(* CODESYS project CtaSysInfluxLog_2.0.0.1.library
   Description: Trendlog Library der CTA
   Version: 2.0.0.1
   Title: CtaSysInfluxLog
   Author: SIS
   DocFormat: reStructuredText
   LanguageModelAttribute: qualified-access-only
   Placeholder: CtaSysInfluxLog
   CompiledLibraryCompatibilityVersion: CODESYS V3.5 SP16 Patch 3
   Company: CTA
   DefaultNamespace: CtaSysInfluxLog

Project tree, tasks and I/O mapping:
  libraries: Standard, 3.5.18.0 (System); VisuSymbols, 4.5.0.0 (System); CtaSysConfig, 2.0.0.0 (CTA); SysFile, 3.5.17.0 (System); SysProcess, 3.5.17.0 (System); StringUtils, 3.5.20.0 (System); CtaVisSymbols, 2.0.0.0 (CTA); CmpIecTask, 3.5.20.50 (System); Common Behaviour Model, 4.0.0.0 (CODESYS); Util, 3.5.19.0 (System); CmpErrors2 Interfaces, * (System); CmpEventMgr, 3.5.17.0 (System); CmpApp, 3.5.17.0 (System); SysDir, 3.5.17.0 (System); SysTypes Interfaces, * (System); CtaAppTime, 1.0.0.1 (CTA)
  40 Visualizations/
    visualisation visInfluxDb
    visualisation visInfluxDbTemp
    visualisation VIS_POPUP_INFLUXDB
  30 Program Organization Units/
    function block FB_INFLUX_LOG [ST]: SendData, FileClose, FileOpen, FileWrite, CreateDataBase, FileDelete, ADD_LOG_NODE, REM_LOG_NODE, DataBuffer, Config, CheckToBigFile, FB_INIT
    NODE/
      BASE/
        function block FB_LOG_NODE [ST]: KEY, VALUE, BIG_SYBIL, ENABLE, SELF, LOW_SYBIL, REGISTER, FB_EXIT, UNREGISTER, LOGTYPE, DESTROY, DESTROYAFTERLOG, UNIXTIME
      STRING/
        function block FB_LOG_NODE_STRING [ST]: SET_VALUE, VALUE, LOGTYPE
      BOOL/
        function block FB_LOG_NODE_BOOL [ST]: VALUE, SET_VALUE, LOGTYPE
      INT/
        function block FB_LOG_NODE_INT [ST]: VALUE, SET_VALUE, LOGTYPE
      REAL/
        function block FB_LOG_NODE_REAL [ST]: VALUE, SET_VALUE, LOGTYPE
    SPACE CATCH/
      function fcSpaceCatch [ST]
    ASYNC SEND/
      function block FB_SEND_ASYNC [ST]: StartAction, SendAction, ResetAction, FB_INIT, DropAction
    FACTORY/
      function block FB_NODE_FACTORY [ST]: GET_BOOL_LOG_NODE, GET_INT_LOG_NODE, GET_REAL_LOG_NODE, GET_STRING_LOG_NODE, READY
    TREND TASK/
      function block FB_TREND_TASK_PROVIDER [ST]: FB_INIT, FB_EXIT, EventCallback
    TASK_SCHEDULER/
      function CYCLIC_TRENDLOG_BACKGROUND_CTA [ST]
      function CYCLIC_TRENDLOG_CTA [ST]
    function GetWorkingDirectory [ST]
  00000000-0000-0000-0000-000000000000|D:\CoDeSys\LibrariesV3\trunk\Intern\CAA\CAA Template\3.4.0.0 draft\Placeholder.xml
  00000000-0000-0000-0000-000000000000|D:\CoDeSys\LibrariesV3\trunk\Intern\CAA\CAA Template\3.2.0.3 draft\Prefix.pdf
  00000000-0000-0000-0000-000000000000|D:\CoDeSys\LibrariesV3\trunk\Intern\CAA\CAA Template\3.5.2.0 draft\Placeholder.xml
  20 Structs/
    data type scParameter
  50 Images/
  10 Documenation/
    global variables VersionHistory
    global variables readMe
  21 Interface/
    interface ITF_LOG_NODE: BIG_SYBIL, KEY, VALUE, ENABLE, SELF, LOGTYPE, LOW_SYBIL, DESTROYAFTERLOG, DESTROY, UNIXTIME
    interface ITF_LOG_NODE_BOOL: SET_VALUE
    interface ITF_LOG_NODE_INT: SET_VALUE
    interface ITF_LOG_NODE_REAL: SET_VALUE
    interface ITF_LOG_NODE_STRING: SET_VALUE
  11 Library Parameter/
  12 Konstanten/
  60 Textlisten/
    text list InfluxStartup
    text list LogState
  13 Globale Variablen/
    global variables GVL_TREND
    global variables GVL_TREND_TASK_PROVIDER
  text list GlobalTextList
  22 Enumeration/
    data type enInfluxDataType
  70 PRG/
*)

// 20 Structs/scParameter
TYPE scParameter :
    STRUCT
       fbServerIp		:	CtaSysConfig.fbSTRING40;
		fbDataBase		:	CtaSysConfig.fbSTRING40;
		fbtLogIntervall	:	CtaSysConfig.fbTIME;
		fbxEnable		:	CtaSysConfig.fbBOOL;
		fbuiPort		:	CtaSysConfig.fbUINT;
    END_STRUCT
END_TYPE

// 22 Enumeration/enInfluxDataType
{attribute 'qualified_only'}
TYPE enInfluxDataType :
(
	TYPE_BOOL 	:= 0,
	TYPE_INT	:= 1,
	TYPE_REAL 	:= 2,
	TYPE_STRING	:= 3	
);
END_TYPE

// 10 Documenation/VersionHistory
(* 

.. image:: ../../Images/CTA_Logo.jpg
   :align: right
   :width: 15% 

**Vorlage**   


============ =========== =========== ============================================
**Date**     **Version** **Author**  **Change**
------------ ----------- ----------- --------------------------------------------
04.03.2021   0.0.0.0     SIS         Vorlage erstellt

============ =========== =========== ============================================


*)
VAR_GLOBAL
    stInfo : STRING:= '0.0.0.0, Vorlage, CTA';
END_VAR

// 10 Documenation/readMe
(*

**ReadMe**

|	**Empfehlung**
|
|	Für das Trendloggen in die InfluxDb wird nachfolgender Code benötigt.                           
|	Zusätzlich muss im PLC_PRG der Fb fbLibAp94_1InfluxDb als Funktionsbaustein Instanziert werden.
|  
|
| *Beispiel* 

 ============= ================================================================================================================================
 Beschreibung  Code                                                                                                
 ============= ================================================================================================================================                   
 Pou oder SmFb .. code-block:: codesys
 
                    // Deklaration der Struktur Variable scInfluxData
                    VAR
                        scInfluxData                    :   WagoAppInfluxDB.typInfluxField;
                    END_VAR     

                    (* Code als actInfluxDb *)
                    // Clear Data
                        scInfluxData.sKey   := '';
                        scInfluxData.sValue := '';
                    // Write Data
                        scInfluxData.sKey   := CONCAT(STR1 := stObjID, STR2 := '_xOn');
                        scInfluxData.sValue := TO_STRING(xOn); 
                        scInfluxData.eType  := WagoAppInfluxDB.eFieldValueType.eFVT_BOOL;
                        LibAp94InfluxDb.gvlLibAp94_1InfluxDb.fbLibAp94_2DataCollecter.proInfluxDbData := scInfluxData;
                    // Clear Data
                        scInfluxData.sKey   := '';
                        scInfluxData.sValue := '';
                    // Write Data
                        scInfluxData.sKey   := CONCAT(STR1 := stObjID, STR2 := '_rOnY');
                        scInfluxData.sValue := TO_STRING(rOnY); 
                        scInfluxData.eType  := WagoAppInfluxDB.eFieldValueType.eFVT_FLOAT;
                        LibAp94InfluxDb.gvlLibAp94_1InfluxDb.fbLibAp94_2DataCollecter.proInfluxDbData := scInfluxData;    
                    // Clear Data
                        scInfluxData.sKey   := '';
                        scInfluxData.sValue := '';
                    // Write Data
                        scInfluxData.sKey   := CONCAT(STR1 := stObjID, STR2 := '_xError');
                        scInfluxData.sValue := TO_STRING(proLockDown); 
                        scInfluxData.eType  := WagoAppInfluxDB.eFieldValueType.eFVT_BOOL;
                        LibAp94InfluxDb.gvlLibAp94_1InfluxDb.fbLibAp94_2DataCollecter.proInfluxDbData := scInfluxData;           
                                                                                                                                                                 
 ============= ================================================================================================================================ 
*)
VAR_GLOBAL
    xReadMeDone              :   BOOL;
END_VAR

// 13 Globale Variablen/GVL_TREND
{attribute 'qualified_only'}
{attribute 'linkalways'}
{attribute 'global_init_slot' := '1000'}
VAR_GLOBAL
	(* ASYNC SEND *)
	ASYNC_SEND				:	FB_SEND_ASYNC;	
	FB_INFLUX_LOG_OBJ		:	FB_INFLUX_LOG;
	FB_INFLUX_NODE_FACTORY	:	FB_NODE_FACTORY;
END_VAR

// 13 Globale Variablen/GVL_TREND_TASK_PROVIDER
{attribute 'qualified_only'}
{attribute 'linkalways'}
{attribute 'global_init_slot' := '1001'}
VAR_GLOBAL
	FB_TREND_TASK_PROVIDER_GLOBAL : FB_TREND_TASK_PROVIDER;	
	dwSEMA_CYCLIC	:	DWORD;				// CYCLIC TASK Semaphore
	dwSEMA_BACK		:	DWORD;				// BACKGRROUND TASK Semaphore
END_VAR

// 21 Interface/ITF_LOG_NODE
INTERFACE ITF_LOG_NODE EXTENDS __SYSTEM.IQueryinterface

PROPERTY BIG_SYBIL : ITF_LOG_NODE
GET
END_GET
SET
END_SET
END_PROPERTY

PROPERTY KEY : STRING(255)
GET
END_GET
SET
END_SET
END_PROPERTY

PROPERTY VALUE : STRING(255)
GET
END_GET
END_PROPERTY

PROPERTY ENABLE : BOOL
SET
END_SET
GET
END_GET
END_PROPERTY

PROPERTY SELF : ITF_LOG_NODE
GET
END_GET
END_PROPERTY

PROPERTY LOGTYPE : enInfluxDataType
GET
END_GET
END_PROPERTY

PROPERTY LOW_SYBIL : ITF_LOG_NODE
GET
END_GET
SET
END_SET
END_PROPERTY

PROPERTY DESTROYAFTERLOG : BOOL
SET
END_SET
GET
END_GET
END_PROPERTY

METHOD INTERNAL DESTROY
VAR_INPUT
END_VAR
END_METHOD

PROPERTY UNIXTIME : ULINT
GET
END_GET
END_PROPERTY

END_INTERFACE

// 30 Program Organization Units/FB_INFLUX_LOG
FUNCTION_BLOCK FB_INFLUX_LOG
VAR
	(* Server Info *)
	UNIXTIME		:	STRING(20);
	(* Log Nodes *)
	_BASE_LOG_NODE	:	ITF_LOG_NODE;
	_TEMP_REG_NODE	:	ITF_LOG_NODE;
	_TEMP_LOG_NODE	:	ITF_LOG_NODE;	
	_TEMP_DES_NODE	:	ITF_LOG_NODE;
	_COUNT			:	UINT;
	(* Case *)
	usiStartUpCase	:	USINT;
	usiLogCase		:	USINT;
	xAbort			:	BOOL;
	(* Buffer *)
	BUFFER			:	STRING(912);
	(* Timers *)
	DELAY			:	Standard.TON	:= (PT := T#20S);
	PULSE			:	Standard.TON	:= (PT := T#1S);
	Fb_TIME			:	CtaAppTime.fbTimeMeasurement;
	ltOut			:	LTIME;
	Fb_TIME_TO_BIG	:	CtaAppTime.fbTimeMeasurement;
	ltOutToBig		:	LTIME;
	xFirstToBig		:	BOOL;
	tCycle			:	TIME;
	taskHandle		:	SysTypes.RTS_IEC_HANDLE;
	pInfo 			: 	POINTER TO CmpIecTask.Task_Info2;	
	(* File Handling *)
	FILE_HANDLE		:	SysFile.RTS_IEC_HANDLE;
	RESULT			:	SysFile.RTS_IEC_RESULT;
	LASTBIGFILESIZE	:	__XWORD;
	FILE_PATH		:	STRING(255);
	(* Config *)
	fbConfigFile	:	CtaSysConfig.fbConfigFile;
	(* Parameter *)
	scParameter		:	scParameter;	
END_VAR
VAR CONSTANT
	COMMA		:	STRING[1] := ',';
	EQUAL		:	STRING[1] := '=';
	SPACE		:	STRING[1] := ' ';
	LINE		:	STRING[1] := '$N';
END_VAR

(* Config *)
Config();
(* Start Up Case *)
CASE usiStartUpCase OF
	0:	(* Delay *)
		DELAY(IN	:= fbConfigFile.proInitDone AND NOT DELAY.Q ,
			  PT	:= T#10S);
		(* Wait *)
		IF DELAY.Q AND scParameter.fbxEnable.proValue THEN
			(*  Get Cycle Time *)
			taskHandle :=  CmpIecTask.IecTaskGetCurrent(ADR(RESULT));
			IF taskHandle <> 0 THEN
				pInfo := CmpIecTask.IecTaskGetInfo3(taskHandle,ADR(RESULT));
				IF pInfo <> 0 THEN
					tCycle := TO_TIME(pInfo^.dwInterval/1000);
				END_IF;		
			END_IF;
			(* SERVER & DATABASE INFO *)
			GVL_TREND.ASYNC_SEND.SERVER 	:= scparameter.fbServerIp.proValue;
			GVL_TREND.ASYNC_SEND.DATABASE 	:= scparameter.fbDataBase.proValue;
			GVL_TREND.ASYNC_SEND.PORT		:= scparameter.fbuiPort.proValue;
			(* Next Case *)
			usiStartUpCase := usiStartUpCase + 1;	
		END_IF;
	1:	(* Create Database *)
		IF CreateDataBase() THEN
			usiStartUpCase := usiStartUpCase + 1;
			usiLogCase   := 1;
		ELSE
			usiStartUpCase := 0;	// Retray with case 0
		END_IF;
	2:	(* Log *)
		CASE usiLogCase OF
			0:
				(* Wait for Database*)
				usiLogCase := usiLogCase + 1;	
				(* ASYNC SEND RESET*)
				GVL_TREND.ASYNC_SEND.Execute := FALSE;		
			1:	
				(* Open File to Save Log *)
				FileOpen();
				usiLogCase := usiLogCase + 1;
			2:	
				(* Log Intervall *)
				PULSE(	IN	:= NOT PULSE.Q,	
						PT	:= LIMIT(T#0MS,scparameter.fbtLogIntervall.proValue - MIN(scparameter.fbtLogIntervall.proValue,(TO_TIME(ltOut)+(tCycle*4)+ T#500MS)),T#10M));

				(* Start Log *)
				IF PULSE.Q OR PULSE.PT = T#0MS THEN
					Fb_TIME.Start();
					UNIXTIME := CONCAT(TO_STRING(Util.GetLocalDateTime(Util.TSW.gc_tzTimeZoneUTC)),'000000');
					(* Get Active Log Data *)
					_COUNT := 0;
					IF __QUERYINTERFACE(_BASE_LOG_NODE,_TEMP_LOG_NODE) THEN
						REPEAT
							(* Check if Valid Log Node *)
							IF __QUERYINTERFACE(_TEMP_LOG_NODE,_TEMP_LOG_NODE) THEN
								(* Buffer Data *)
								DataBuffer(_TEMP_LOG_NODE.KEY,_TEMP_LOG_NODE.VALUE,_TEMP_LOG_NODE.DESTROYAFTERLOG,TO_STRING(_TEMP_LOG_NODE.UNIXTIME));
								(* COUNT *)
								_COUNT := _COUNT + 1;
								(* Get Next Log Node *)
								_TEMP_DES_NODE := _TEMP_LOG_NODE;
								_TEMP_LOG_NODE := _TEMP_LOG_NODE.LOW_SYBIL;
								(* Destroy if no longer needed *)
								IF _TEMP_DES_NODE.DESTROYAFTERLOG THEN
									_TEMP_DES_NODE.DESTROY();
									_TEMP_DES_NODE := 0;
								END_IF;
							END_IF;
						(* End Repeat if no more Node *)
						UNTIL NOT __QUERYINTERFACE(_TEMP_LOG_NODE,_TEMP_LOG_NODE)
						END_REPEAT
					END_IF;
					(* Check if unwritet Buffer needs write *)
					IF Stu.StrLenA(ADR(BUFFER)) > 0 THEN
						FileWrite();
						BUFFER := '';
					END_IF;
					(* Get Time *)
					ltOut := Fb_TIME.Stop();
					(* Next Case Step *)
					usiLogCase := usiLogCase + 1;
				END_IF;
			3:
				(* Reset if Failed *)
				IF GVL_TREND.ASYNC_SEND._RESULT <> CmpErrors.Errors.ERR_OK THEN
					GVL_TREND.ASYNC_SEND.ResetAction();
				END_IF;
				(* Close File *)
				IF NOT GVL_TREND.ASYNC_SEND.Busy AND NOT GVL_TREND.ASYNC_SEND.Execute THEN
					FileClose();	
					IF FILE_HANDLE = 0 THEN
						GVL_TREND.ASYNC_SEND.Execute := TRUE;	
					END_IF;
				END_IF;
								
				(* Get Condition *)
				IF GVL_TREND.ASYNC_SEND.Done THEN	
					(* Send Data Ok *)
					IF GVL_TREND.ASYNC_SEND.xSendOk THEN
						(* Delete after Sending *)
						FileDelete();
						xFirstToBig	:= FALSE;
					ELSIF GVL_TREND.ASYNC_SEND.Drop THEN
						(* Create new Db after Drop and delete file*)
						FileDelete();
						usiStartUpCase := 0;
					ELSE
						(* Time To Big *)
						IF NOT xFirstToBig THEN
							Fb_TIME_TO_BIG.Start();
							xFirstToBig := TRUE;
						END_IF;
						(* Check if File is to Big if not Sendet*)
						IF CheckToBigFile() THEN
							(* Delete if to Big *)
							FileDelete();	
							usiStartUpCase := 0;
							
							(* To Big Time *)
							ltOutToBig := Fb_TIME_TO_BIG.Stop();
							xFirstToBig := FALSE;
						END_IF;
					END_IF;
					IF NOT xAbort THEN
						(* Return to 1 *)
						usiLogCase   := 1;	
						(* ASYNC SEND RESET*)
						GVL_TREND.ASYNC_SEND.Execute := FALSE;			
					ELSE
						(* Restart *)
						xAbort := FALSE;
						usiStartUpCase	:= 0;
						usiLogCase      := 0;
					END_IF;	
				END_IF;
			ELSE
				(* Return to 1 if Case overflow *)
				usiLogCase := 1;	
			END_CASE;
	ELSE
		(* Return to 0 if Case overflow *)
		usiStartUpCase 	:= 0;
		usiLogCase		:= 0;
END_CASE;

METHOD SendData : BOOL
VAR_INPUT
END_VAR
VAR
	_COMMAND	:	STRING(255);
	_RESPONS	:	STRING(255);
	_RESULT		:	SysTypes.RTS_IEC_RESULT;
END_VAR





//COMMAND	:= 'curl -i -XPOST --data-binary @/home/codesys_root/PlcLogic/trend/InfluxDb.txt http://10.0.1.22:8086/write?db=CtaInfluxDb';
END_METHOD

METHOD FileClose : BOOL
VAR_INPUT
END_VAR
IF FILE_HANDLE <> 0 THEN
	__TRY
		SysFile.SysFileClose(FILE_HANDLE);
		FILE_HANDLE := 0;
	__CATCH
		;
	__ENDTRY;
END_IF;
END_METHOD

METHOD FileOpen : BOOL
VAR_INPUT
END_VAR
IF FILE_HANDLE = 0 THEN
	FILE_HANDLE := SysFile.SysFileOpen(FILE_PATH,SysFile.ACCESS_MODE.AM_APPEND_PLUS,ADR(RESULT));
END_IF;
END_METHOD

METHOD FileWrite : BOOL
VAR
END_VAR
IF FILE_HANDLE <> 0 THEN
	(* Write *)
	__TRY
		SysFile.SysFileWrite(FILE_HANDLE,ADR(BUFFER),TO___XWORD(Stu.StrLenA(ADR(BUFFER))),ADR(RESULT));
	__CATCH
		;
	__ENDTRY
END_IF;
END_METHOD

METHOD CreateDataBase : BOOL
VAR_INPUT
END_VAR
VAR
	COMMAND	:	STRING(255);
	RESPONS	:	STRING(255);	
END_VAR
COMMAND	:= 	Standard.CONCAT(
			Standard.CONCAT(
			Standard.CONCAT(
			Standard.CONCAT(
			Standard.CONCAT(
			Standard.CONCAT(
							'curl -i -XPOST --connect-timeout 5 $'http://',
							GVL_TREND.ASYNC_SEND.SERVER),
							':'),
							TO_STRING(GVL_TREND.ASYNC_SEND.PORT)),
							'/query?u=CTA&p=CtaInfluxDb$' --data-urlencode $'q=CREATE DATABASE "'),
							GVL_TREND.ASYNC_SEND.DATABASE),
							'"$' epoch="ms"');
(* Create Database *)
SysProcess_Implementation.SysProcessExecuteCommand2(COMMAND,RESPONS,SIZEOF(RESPONS),ADR(RESULT));
(* Get Error *)
IF Standard.FIND(RESPONS,'error') = 0 AND Standard.FIND(RESPONS,'Error') = 0 AND RESPONS <> '' THEN
	CreateDataBase := TRUE;
END_IF;
END_METHOD

METHOD FileDelete : BOOL
VAR_INPUT
END_VAR
IF FILE_HANDLE = 0 THEN
	SysFile.SysFileDelete(FILE_PATH);
END_IF;
END_METHOD

METHOD ADD_LOG_NODE
VAR_INPUT
	ITF_LOG_NODE_IN	:	ITF_LOG_NODE;
END_VAR
IF __QUERYINTERFACE(_BASE_LOG_NODE,_BASE_LOG_NODE) THEN
	IF __QUERYINTERFACE(_TEMP_REG_NODE,_TEMP_REG_NODE) THEN
		_TEMP_REG_NODE.LOW_SYBIL := ITF_LOG_NODE_IN;
		_TEMP_REG_NODE := ITF_LOG_NODE_IN;
	ELSE
		_TEMP_REG_NODE := ITF_LOG_NODE_IN;
		_BASE_LOG_NODE.LOW_SYBIL := ITF_LOG_NODE_IN;
	END_IF;		
ELSE
	_BASE_LOG_NODE := ITF_LOG_NODE_IN;
END_IF;
END_METHOD

METHOD REM_LOG_NODE 
VAR_INPUT
	ITF_LOG_NODE_IN	:	ITF_LOG_NODE;
END_VAR
VAR
	_ITF_BIG_SYBIL	:	ITF_LOG_NODE;
	_ITF_LOW_SYBIL	:	ITF_LOG_NODE;
END_VAR
IF __QUERYINTERFACE(ITF_LOG_NODE_IN,ITF_LOG_NODE_IN) THEN
	(* GET SYBIL *)
	_ITF_BIG_SYBIL := ITF_LOG_NODE_IN.BIG_SYBIL;
	_ITF_LOW_SYBIL := ITF_LOG_NODE_IN.LOW_SYBIL;
	(* Check if BASE LOG Node *)
	IF ITF_LOG_NODE_IN = _BASE_LOG_NODE THEN
		IF __QUERYINTERFACE(_ITF_LOW_SYBIL,_ITF_LOW_SYBIL) THEN
			_BASE_LOG_NODE := _ITF_LOW_SYBIL;
		ELSE
			_BASE_LOG_NODE := 0;
		END_IF;
	END_IF;
	(* Check if Temp REG Node *)
	IF ITF_LOG_NODE_IN = _TEMP_REG_NODE THEN
		IF __QUERYINTERFACE(_ITF_BIG_SYBIL,_ITF_BIG_SYBIL) THEN
			_TEMP_REG_NODE := _ITF_BIG_SYBIL;
		ELSE
			_TEMP_REG_NODE := 0;
		END_IF;
	END_IF;
	(* Give BIG SIBIL To LOW SYBIL *)
	IF __QUERYINTERFACE(_ITF_BIG_SYBIL,_ITF_BIG_SYBIL) THEN
		_ITF_BIG_SYBIL.LOW_SYBIL := _ITF_LOW_SYBIL;
	END_IF;
	(* Give LOW SIBIL To BIG SYBIL *)
	IF __QUERYINTERFACE(_ITF_LOW_SYBIL,_ITF_LOW_SYBIL) THEN
		_ITF_LOW_SYBIL.BIG_SYBIL := _ITF_BIG_SYBIL;
	END_IF;
	(* CLEAR *)
	ITF_LOG_NODE_IN.BIG_SYBIL := 0;
	ITF_LOG_NODE_IN.LOW_SYBIL := 0;
END_IF;
END_METHOD

METHOD DataBuffer : BOOL
VAR_INPUT
	KEY					:	STRING(255);
	VALUE				:	STRING(255);
	DESTROY				:	BOOL;
	UNIXTIME_DESTROY	:	STRING(20)	:= UNIXTIME;
END_VAR
IF FILE_HANDLE <> 0 THEN
	IF KEY <> '' AND VALUE <> '' THEN		
		(* DATABASE *)
		Stu.StrConcatA(ADR(GVL_TREND.ASYNC_SEND.DATABASE),ADR(BUFFER),TO_INT(SIZEOF(BUFFER)));
		(* SPACE *)
		Stu.StrConcatA(ADR(SPACE),ADR(BUFFER),TO_INT(SIZEOF(BUFFER)));
		(* KEY *) 
		Stu.StrConcatA(ADR(KEY),ADR(BUFFER),TO_INT(SIZEOF(BUFFER)));	
		(* EQUAL *)
		Stu.StrConcatA(ADR(EQUAL),ADR(BUFFER),TO_INT(SIZEOF(BUFFER)));
		(* VALUE *)
		Stu.StrConcatA(ADR(VALUE),ADR(BUFFER),TO_INT(SIZEOF(BUFFER)));
		(* SPACE *)
		Stu.StrConcatA(ADR(SPACE),ADR(BUFFER),TO_INT(SIZEOF(BUFFER)));		
		(* UNIX *)
		IF DESTROY THEN
			Stu.StrConcatA(ADR(UNIXTIME_DESTROY),ADR(BUFFER),TO_INT(SIZEOF(BUFFER)));	
		ELSE
			Stu.StrConcatA(ADR(UNIXTIME),ADR(BUFFER),TO_INT(SIZEOF(BUFFER)));	
		END_IF;
		(* NEW LINE *)
		Stu.StrConcatA(ADR(LINE),ADR(BUFFER),TO_INT(SIZEOF(BUFFER)));	
		(* Store If Buffer is Full *)
		IF SIZEOF(BUFFER) - TO_UINT(Stu.StrLenA(ADR(BUFFER))) <= 574 THEN
			FileWrite();
			BUFFER := '';
		END_IF;			
	END_IF;
END_IF;
END_METHOD

ACTION Config:
fbConfigFile();
scparameter.fbServerIp		(_usiParaNr := 1,	itfConfigFb := fbConfigFile,_WertInit := '10.0.1.12');
scparameter.fbDataBase		(_usiParaNr := 2,	itfConfigFb := fbConfigFile,_WertInit := 'CtaInfluxDb');
scparameter.fbtLogIntervall	(_usiParaNr := 3,	itfConfigFb := fbConfigFile,_WertInit := T#2S	,	_MinInit	:= T#1S,	_MaxInit := T#1D);
scparameter.fbxEnable		(_usiParaNr := 4,	itfConfigFb := fbConfigFile,_WertInit := TRUE	);
scparameter.fbuiPort		(_usiParaNr := 5,	itfConfigFb := fbConfigFile,_WertInit := 8086	);

(* Server Adress *)
IF scparameter.fbxEnable.proStateChanged THEN
	xAbort := TRUE;
END_IF;
(* Server Adress *)
IF scparameter.fbServerIp.proStateChanged THEN
	xAbort := TRUE;
END_IF;
(* Database Name *)
IF scparameter.fbDataBase.proStateChanged THEN
	xAbort := TRUe;
END_IF;
(* Port *)
IF scparameter.fbuiPort.proStateChanged THEN
	xAbort := TRUE;
END_IF;
END_ACTION

METHOD CheckToBigFile : BOOL
VAR_INPUT
END_VAR
LASTBIGFILESIZE := SysFile.SysFileGetSize(FILE_PATH,ADR(RESULT));
IF LASTBIGFILESIZE >= 25000000 THEN
	CheckToBigFile := TRUE;
ELSE
	CheckToBigFile := FALSE;
END_IF;
END_METHOD

//FB_Init ist immer implizit verfügbar und wird primär für die Initialisierung verwendet.
//Der Rückgabewert wird nicht ausgewertet. Für gezielte Einflussnahme können Sie
//die Methoden explizit deklarieren und darin mit dem Standard-Initialisierungscode 
//zusätzlichen Code bereitstellen. Sie können den Rückgabewert auswerten.
METHOD FB_Init: BOOL
VAR_INPUT    
bInitRetains: BOOL; // TRUE: Die Retain-Variablen werden initialisiert (Reset warm / Reset kalt)    
bInCopyCode: BOOL;  // TRUE: Die Instanz wird danach in den Kopiercode kopiert (Online-Change)
END_VAR
FILE_PATH := Standard.CONCAT(GetWorkingDirectory(),'/trend/InfluxDb.txt');
END_METHOD

END_FUNCTION_BLOCK

// 30 Program Organization Units/GetWorkingDirectory
FUNCTION GetWorkingDirectory : String(255)
VAR_INPUT
END_VAR
VAR
	RTS_IEC_RESULT : SysTypes.RTS_IEC_RESULT;
END_VAR

SysDir.SysDirGetCurrent(GetWorkingDirectory,SIZEOF(GetWorkingDirectory));

END_FUNCTION

// 30 Program Organization Units/NODE/BASE/FB_LOG_NODE
{attribute 'enable_dynamic_creation'}
FUNCTION_BLOCK FB_LOG_NODE IMPLEMENTS ITF_LOG_NODE
VAR_INPUT
END_VAR
VAR_OUTPUT
END_VAR
VAR
	xEnable				:	BOOL;
	xEnableOld			:	BOOL;
	xDestroyAfterLog	:	BOOL;
	uliUnixTime			:	ULINT;
	stKey				:	STRING(255);	
	_ITF_BIG_SYBIL		:	ITF_LOG_NODE;
	_ITF_LOW_SYBIL		:	ITF_LOG_NODE;
END_VAR

PROPERTY FINAL KEY : STRING(255)
GET
KEY := stKey;
END_GET
SET
stKEy := fcSpaceCatch(KEY);
END_SET
END_PROPERTY

PROPERTY VALUE : STRING(255)
GET
VALUE := '';
END_GET
END_PROPERTY

{attribute 'estimated-stack-usage' := '104'}
PROPERTY FINAL BIG_SYBIL : ITF_LOG_NODE
GET
BIG_SYBIL := _ITF_BIG_SYBIL;
END_GET
SET
_ITF_BIG_SYBIL := BIG_SYBIL;
IF __QUERYINTERFACE(_ITF_BIG_SYBIL,_ITF_BIG_SYBIL) THEN
	IF _ITF_BIG_SYBIL.LOW_SYBIL <> SELF THEN
		_ITF_BIG_SYBIL.LOW_SYBIL := THIS^;
	END_IF;
END_IF;
END_SET
END_PROPERTY

PROPERTY FINAL ENABLE : BOOL
GET
ENABLE := xEnable;
END_GET
SET
xEnable := ENABLE;
IF xEnable <> xEnableOld THEN
	xEnableOld := xEnable;
	IF NOT xEnable THEN
		DESTROY();
	ELSE
		REGISTER();
	END_IF;
END_IF;
END_SET
END_PROPERTY

PROPERTY FINAL SELF : ITF_LOG_NODE
GET
SELF := THIS^;
END_GET
END_PROPERTY

{attribute 'estimated-stack-usage' := '104'}
PROPERTY FINAL LOW_SYBIL : ITF_LOG_NODE
GET
LOW_SYBIL := _ITF_LOW_SYBIL;
END_GET
SET
_ITF_LOW_SYBIL := LOW_SYBIL;
IF __QUERYINTERFACE(_ITF_LOW_SYBIL,_ITF_LOW_SYBIL) THEN
	IF _ITF_LOW_SYBIL.BIG_SYBIL <> SELF THEN
		_ITF_LOW_SYBIL.BIG_SYBIL := THIS^;
	END_IF;
END_IF;
END_SET
END_PROPERTY

METHOD FINAL REGISTER : BOOL
VAR_INPUT
END_VAR
GVL_TREND.FB_INFLUX_LOG_OBJ.ADD_LOG_NODE(THIS^);
END_METHOD

//FB_Exit muss explizit implementiert werden. Wenn es eine Implementierung gibt, dann wird 
//die Methode aufgerufen, bevor die Steuerung den Code der Funktionsbaustein-Instanz entfernt
//(impliziter Aufruf. Der Rückgabewert wird nicht ausgewertet.
METHOD FB_Exit: BOOL
VAR_INPUT    
bInCopyCode: BOOL;  // TRUE: Die Exit-Methode wird aufgerufen, um die Instanz zu verlassen, die hinterher kopiert wird Online-Change).  
END_VAR
IF NOT bInCopyCode THEN
	UNREGISTER();
END_IF;
END_METHOD

METHOD FINAL UNREGISTER : BOOL
VAR_INPUT
END_VAR
GVL_TREND.FB_INFLUX_LOG_OBJ.REM_LOG_NODE(THIS^);
END_METHOD

PROPERTY LOGTYPE : enInfluxDataType
GET
LOGTYPE := enInfluxDataType.TYPE_STRING;
END_GET
END_PROPERTY

METHOD DESTROY
VAR_INPUT
END_VAR
VAR
	_SELF_POINTER	:	POINTER TO FB_LOG_NODE;
END_VAR
UNREGISTER();
_SELF_POINTER := THIS;
__DELETE(_SELF_POINTER);
END_METHOD

PROPERTY DESTROYAFTERLOG : BOOL
SET
xDestroyAfterLog := DESTROYAFTERLOG;
IF xDestroyAfterLog AND uliUnixTime = 0 THEN
	uliUnixTime := TO_ULINT(CONCAT(TO_STRING(Util.GetLocalDateTime(Util.TSW.gc_tzTimeZoneUTC)),'000000'));
END_IF;
END_SET
GET
DESTROYAFTERLOG := xDestroyAfterLog;
END_GET
END_PROPERTY

PROPERTY UNIXTIME : ULINT
GET
UNIXTIME := uliUnixTime;
END_GET
END_PROPERTY

END_FUNCTION_BLOCK

// 30 Program Organization Units/SPACE CATCH/fcSpaceCatch
FUNCTION fcSpaceCatch : STRING
VAR_INPUT
	stIn	: STRING;
END_VAR
VAR
	usiSafe	:	USINT;
END_VAR

fcSpaceCatch := stIn;
WHILE Standard.FIND(fcSpaceCatch,' ') > 0 AND usiSafe < 81 DO
	fcSpaceCatch := Standard.REPLACE(fcSpaceCatch,'_',1,Standard.FIND(fcSpaceCatch,' '));
	usiSafe := usiSafe + 1;
END_WHILE;

END_FUNCTION

// 30 Program Organization Units/NODE/STRING/FB_LOG_NODE_STRING
{attribute 'enable_dynamic_creation'}
FUNCTION_BLOCK FB_LOG_NODE_STRING EXTENDS FB_LOG_NODE IMPLEMENTS ITF_LOG_NODE_STRING
VAR
	stValue	:	STRING(250);
END_VAR;

PROPERTY SET_VALUE : STRING(255)
SET
stValue := SET_VALUE;
END_SET
END_PROPERTY

PROPERTY VALUE : STRING(255)
GET
IF stValue <> '' THEN
	VALUE := CONCAT(CONCAT('"',stValue),'"');
ELSE
	VALUE := '';
END_IF;
END_GET
END_PROPERTY

PROPERTY LOGTYPE : enInfluxDataType
GET
LOGTYPE := enInfluxDataType.TYPE_STRING;
END_GET
END_PROPERTY

END_FUNCTION_BLOCK

// 21 Interface/ITF_LOG_NODE_STRING
INTERFACE ITF_LOG_NODE_STRING EXTENDS ITF_LOG_NODE

PROPERTY SET_VALUE : STRING(255)
SET
END_SET
END_PROPERTY

END_INTERFACE

// 30 Program Organization Units/NODE/BOOL/FB_LOG_NODE_BOOL
{attribute 'enable_dynamic_creation'}
FUNCTION_BLOCK FB_LOG_NODE_BOOL EXTENDS FB_LOG_NODE IMPLEMENTS ITF_LOG_NODE_BOOL
VAR
	xValue	:	BOOL;
END_VAR

PROPERTY VALUE : STRING(255)
GET
VALUE := TO_STRING(xValue);
END_GET
END_PROPERTY

PROPERTY SET_VALUE : BOOL
SET
xValue := SET_VALUE;
END_SET
END_PROPERTY

PROPERTY LOGTYPE : enInfluxDataType
GET
LOGTYPE := enInfluxDataType.TYPE_BOOL;
END_GET
END_PROPERTY

END_FUNCTION_BLOCK

// 21 Interface/ITF_LOG_NODE_BOOL
INTERFACE ITF_LOG_NODE_BOOL EXTENDS ITF_LOG_NODE

PROPERTY SET_VALUE : BOOL
SET
END_SET
END_PROPERTY

END_INTERFACE

// 30 Program Organization Units/NODE/INT/FB_LOG_NODE_INT
{attribute 'enable_dynamic_creation'}
FUNCTION_BLOCK FB_LOG_NODE_INT EXTENDS FB_LOG_NODE IMPLEMENTS ITF_LOG_NODE_INT
VAR
	iValue	:	INT;
END_VAR

PROPERTY VALUE : STRING(255)
GET
VALUE := CONCAT(TO_STRING(iValue),'i');
END_GET
END_PROPERTY

PROPERTY SET_VALUE : INT
SET
iValue := SET_VALUE;
END_SET
END_PROPERTY

PROPERTY LOGTYPE : enInfluxDataType
GET
LOGTYPE := enInfluxDataType.TYPE_INT;
END_GET
END_PROPERTY

END_FUNCTION_BLOCK

// 21 Interface/ITF_LOG_NODE_INT
INTERFACE ITF_LOG_NODE_INT EXTENDS ITF_LOG_NODE

PROPERTY SET_VALUE : INT
SET
END_SET
END_PROPERTY

END_INTERFACE

// 30 Program Organization Units/NODE/REAL/FB_LOG_NODE_REAL
{attribute 'enable_dynamic_creation'}
FUNCTION_BLOCK FB_LOG_NODE_REAL EXTENDS FB_LOG_NODE IMPLEMENTS ITF_LOG_NODE_REAL
VAR
	rValue	:	REAL;
END_VAR

PROPERTY VALUE : STRING(255)
GET
VALUE := TO_STRING(rValue);
END_GET
END_PROPERTY

PROPERTY SET_VALUE : REAL
SET
rValue := SET_VALUE;
END_SET
END_PROPERTY

PROPERTY LOGTYPE : enInfluxDataType
GET
LOGTYPE := enInfluxDataType.TYPE_REAL;
END_GET
END_PROPERTY

END_FUNCTION_BLOCK

// 21 Interface/ITF_LOG_NODE_REAL
INTERFACE ITF_LOG_NODE_REAL EXTENDS ITF_LOG_NODE

PROPERTY SET_VALUE : REAL
SET
END_SET
END_PROPERTY

END_INTERFACE

// 30 Program Organization Units/ASYNC SEND/FB_SEND_ASYNC
FUNCTION_BLOCK FB_SEND_ASYNC 
VAR_INPUT
	Execute			:	BOOL;
	SERVER			:	STRING(40)	:= '0.0.0.0';
	DATABASE		:	STRING(40)	:= 'CtaInfluxDb';
	PORT			:	UINT		:= 8086;
END_VAR
VAR_OUTPUT
	Done			:	BOOL;
	Busy			:	BOOL;
	Drop			:	BOOL;
	_RESULT			:	SysTypes.RTS_IEC_RESULT;
	xSendOk			:	BOOL;
END_VAR
VAR
	ExecuteTemp	:	BOOL;
	_COMMAND	:	STRING(255);
	_RESPONS	:	STRING(255);	
	FILE_PATH	:	STRING(255);
END_VAR

ExecuteTemp := Execute;
IF ExecuteTemp AND NOT Busy AND NOT Done THEN
	Busy := TRUE;
	IF StartAction() THEN
		IF SendAction() THEN
			Busy := FALSE;
			Done := TRUE;
		END_IF;
	END_IF;
ELSIF NOT ExecuteTemp THEN
	Busy 	:= FALSE;
	Done 	:= FALSE;
	xSendOk := FALSE;
END_IF;

METHOD StartAction : BOOL;
_COMMAND:= 	Standard.CONCAT(
			Standard.CONCAT(
			Standard.CONCAT(
			Standard.CONCAT(
			Standard.CONCAT(
			Standard.CONCAT(
			Standard.CONCAT(
							'curl -i -XPOST --connect-timeout 2 --data-binary @',
							FILE_PATH),
							' http://'),
							SERVER),
							':'),
							TO_STRING(PORT)),
							'/write?db='),
							DATABASE);
StartAction := TRUE;
END_METHOD

METHOD SendAction : BOOL
VAR
	start_pos	:	INT;
	lenght		:	INT;
	temp_string	:	STRING(255);
END_VAR
	(* Send Data *)
	__TRY
		SysProcess_Implementation.SysProcessExecuteCommand2(_COMMAND,_RESPONS,SIZEOF(_RESPONS),ADR(_RESULT));
	__CATCH
		xSendOk   := FALSE;
	__ENDTRY
	
	(* Get Error *)
	IF Standard.FIND(_RESPONS,'204 No Content') > 0 THEN
		xSendOk   := TRUE;
		Drop      := FALSE;
	ELSIF (Standard.FIND(_RESPONS,'400 Bad Request') > 0 AND Standard.FIND(_RESPONS,'field type conflict') > 0) OR (Standard.FIND(_RESPONS,'500 Internal Server Error') > 0 AND Standard.FIND(_RESPONS,'Influxdb-Error') > 0) THEN
		DropAction();
		Drop      := TRUE;
		xSendOk   := FALSE;
	ELSE
		xSendOk   := FALSE;
	END_IF;
	
	SendAction := TRUE;
END_METHOD

(* The ``ResetAction`` is running until the output ``xComplete`` is ``TRUE``.
 If ``xComplete`` is ``TRUE`` the state |STATE.DORMANT| is reached.*)
METHOD ResetAction
VAR
	RESETCOMAND	:	STRING;
END_VAR
(* Send Data *)
__TRY
	RESETCOMAND	:= '\x03';
	SysProcess_Implementation.SysProcessExecuteCommand(RESETCOMAND,ADR(_RESULT));
__CATCH
	Done	:= TRUE;
	Drop    := FALSE;
	Busy 	:= FALSE;
	_RESULT := 0;
__ENDTRY
END_METHOD

//FB_Init ist immer implizit verfügbar und wird primär für die Initialisierung verwendet.
//Der Rückgabewert wird nicht ausgewertet. Für gezielte Einflussnahme können Sie
//die Methoden explizit deklarieren und darin mit dem Standard-Initialisierungscode 
//zusätzlichen Code bereitstellen. Sie können den Rückgabewert auswerten.
METHOD FB_Init: BOOL
VAR_INPUT    
bInitRetains: BOOL; // TRUE: Die Retain-Variablen werden initialisiert (Reset warm / Reset kalt)    
bInCopyCode: BOOL;  // TRUE: Die Instanz wird danach in den Kopiercode kopiert (Online-Change)
END_VAR
FILE_PATH := Standard.CONCAT(GetWorkingDirectory(),'/trend/InfluxDb.txt');
END_METHOD

METHOD DropAction
_COMMAND:= 	Standard.CONCAT(
			Standard.CONCAT(
			Standard.CONCAT(
			Standard.CONCAT(
			Standard.CONCAT(
			Standard.CONCAT(
			Standard.CONCAT(
			Standard.CONCAT(
			Standard.CONCAT(
							'curl -i -XPOST http://',
							SERVER),
							':'),
							TO_STRING(PORT)),
							'/query --data-urlencode $'db='),
							DATABASE),
							'$' '),
							'--data-urlencode $'q=DROP DATABASE '),
							DATABASE),
							'$'');
	__TRY
		SysProcess_Implementation.SysProcessExecuteCommand2(_COMMAND,_RESPONS,SIZEOF(_RESPONS),ADR(_RESULT));
	__CATCH
		xSendOk   	:= FALSE;
	__ENDTRY
END_METHOD

END_FUNCTION_BLOCK

// 30 Program Organization Units/FACTORY/FB_NODE_FACTORY
FUNCTION_BLOCK FB_NODE_FACTORY
VAR_INPUT
END_VAR
VAR_OUTPUT
	udiMissingBoolMemory		:	UDINT;
	udiMissingIntMemory			:	UDINT;
	udiMissingRealMemory		:	UDINT;
	udiMissingStringMemory		:	UDINT;
END_VAR
VAR
	dwSemaBool					:	DWORD;
	dwSemaInt					:	DWORD;
	dwSemaReal					:	DWORD;
	dwSemaString				:	DWORD;
END_VAR

METHOD GET_BOOL_LOG_NODE : ITF_LOG_NODE_BOOL;
VAR_OUTPUT
	xSema		:	BOOL;
END_VAR
VAR
	pTempNode	:	POINTER TO FB_LOG_NODE_BOOL;
	dwCurrent	:	DWORD;
END_VAR
dwCurrent := TEST_AND_SET(dwSemaBool);
IF dwCurrent = 0 THEN
	IF udiMissingBoolMemory = 0 THEN
		pTempNode := __NEW(FB_LOG_NODE_BOOL);
		IF pTempNode <> 0 THEN
			GET_BOOL_LOG_NODE := pTempNode^;
			pTempNode := 0;
		ELSE
			GET_BOOL_LOG_NODE := 0;
			udiMissingBoolMemory := udiMissingBoolMemory + SIZEOF(FB_LOG_NODE_BOOL);
		END_IF;
	ELSE
		udiMissingBoolMemory := udiMissingBoolMemory + SIZEOF(FB_LOG_NODE_BOOL);
	END_IF;
	dwSemaBool := 0;
ELSE
	xSema := TRUE;
END_IF;
END_METHOD

METHOD GET_INT_LOG_NODE : ITF_LOG_NODE_INT;
VAR_OUTPUT
	xSema		:	BOOL;
END_VAR
VAR
	pTempNode	:	POINTER TO FB_LOG_NODE_INT;
	dwCurrent	:	DWORD;
END_VAR
dwCurrent := TEST_AND_SET(dwSemaInt);
IF dwCurrent = 0 THEN
	IF udiMissingIntMemory = 0 THEN
		pTempNode := __NEW(FB_LOG_NODE_INT);
		IF pTempNode <> 0 THEN
			GET_INT_LOG_NODE := pTempNode^;
			pTempNode := 0;
		ELSE
			GET_INT_LOG_NODE := 0;
			udiMissingIntMemory := udiMissingIntMemory + SIZEOF(FB_LOG_NODE_INT);
		END_IF;
	ELSE
		udiMissingIntMemory := udiMissingIntMemory + SIZEOF(FB_LOG_NODE_INT);
	END_IF;
	dwSemaInt := 0;
ELSE
	xSema := TRUE;
END_IF;
END_METHOD

METHOD GET_REAL_LOG_NODE : ITF_LOG_NODE_REAL;
VAR_OUTPUT
	xSema		:	BOOL;
END_VAR
VAR
	pTempNode	:	POINTER TO FB_LOG_NODE_REAL;
	dwCurrent	:	DWORD;
END_VAR
dwCurrent := TEST_AND_SET(dwSemaReal);
IF dwCurrent = 0 THEN 
	IF udiMissingRealMemory = 0 THEN
		pTempNode := __NEW(FB_LOG_NODE_REAL);
		IF pTempNode <> 0 THEN
			GET_REAL_LOG_NODE := pTempNode^;
			pTempNode := 0;
		ELSE
			GET_REAL_LOG_NODE := 0;
			udiMissingRealMemory := udiMissingRealMemory + SIZEOF(FB_LOG_NODE_REAL);
		END_IF;
	ELSE
		udiMissingRealMemory := udiMissingRealMemory + SIZEOF(FB_LOG_NODE_REAL);
	END_IF;
	dwSemaReal := 0;
ELSE
	xSema := TRUE;
END_IF;
END_METHOD

METHOD GET_STRING_LOG_NODE : ITF_LOG_NODE_STRING;
VAR_OUTPUT
	xSema		:	BOOL;
END_VAR
VAR
	pTempNode	:	POINTER TO FB_LOG_NODE_STRING;
	dwCurrent	:	DWORD;
END_VAR
dwCurrent := TEST_AND_SET(dwSemaString);
IF dwCurrent = 0 THEN 
	IF udiMissingStringMemory = 0 THEN
		pTempNode := __NEW(FB_LOG_NODE_STRING);
		IF pTempNode <> 0 THEN
			GET_STRING_LOG_NODE := pTempNode^;
			pTempNode := 0;
		ELSE
			GET_STRING_LOG_NODE := 0;
			udiMissingStringMemory := udiMissingStringMemory + SIZEOF(FB_LOG_NODE_STRING);
		END_IF;
	ELSE
		udiMissingStringMemory := udiMissingStringMemory + SIZEOF(FB_LOG_NODE_STRING);	
	END_IF;
	dwSemaString := 0;
ELSE
	xSema := TRUE;
END_IF;
END_METHOD

PROPERTY READY : BOOL
GET
READY := TRUE;
END_GET
END_PROPERTY

END_FUNCTION_BLOCK

// 30 Program Organization Units/TREND TASK/FB_TREND_TASK_PROVIDER
FUNCTION_BLOCK FB_TREND_TASK_PROVIDER IMPLEMENTS CmpEventMgr.ICmpEventCallback
VAR_INPUT
END_VAR
VAR_OUTPUT
END_VAR
VAR
	(* Application *)
	APPLICATION_THIS					:	POINTER TO CmpIecTask.APPLICATION;
	RESULT_APPLICATION_THIS				:	SysTypes.RTS_IEC_RESULT;
	(* EVENT HANDLER *)             		
	HANDLE_EVENT_COM_CYCLE				:	SysTypes.RTS_IEC_HANDLE;
	HANDLE_CALBACK						:	SysTypes.RTS_IEC_HANDLE;
	
	(* CYCLIC_TIME_BACKGROUND_CTA *)
	INFO_CYCLIC_TRENDLOG_BACKGROUND		:	CmpIecTask.Task_Info2;
	NAME_CYCLIC_TRENDLOG_BACKGROUND		:	STRING := 'CYCLIC_TRENDLOG_BACKGROUND_CTA';	
	HANDLE_CYCLIC_TRENDLOG_BACKGROUND	:	SysTypes.RTS_IEC_HANDLE;
	RESULT_CYCLIC_TRENDLOG_BACKGROUND	:	SysTypes.RTS_IEC_RESULT;	

	(* CYCLIC_TRENDDLOG_CTA *)
	INFO_CYCLIC_TRENDLOG				:	CmpIecTask.Task_Info2;
	NAME_CYCLIC_TRENDLOG				:	STRING := 'CYCLIC_TRENDLOG_CTA';	
	HANDLE_CYCLIC_TRENDLOG				:	SysTypes.RTS_IEC_HANDLE;
	RESULT_CYCLIC_TRENDLOG				:	SysTypes.RTS_IEC_RESULT;	
		
	(* HELPER *)
	CYCLIC_TYPE							:	DWORD	:= 11;	
	EMPTY_STRING						:	STRING(1);
	TEMP_TASK_INFO						:	POINTER TO CmpIecTask.Task_Info2;
		 
END_VAR

//FB_Init ist immer implizit verfügbar und wird primär für die Initialisierung verwendet.
//Der Rückgabewert wird nicht ausgewertet. Für gezielte Einflussnahme können Sie
//die Methoden explizit deklarieren und darin mit dem Standard-Initialisierungscode 
//zusätzlichen Code bereitstellen. Sie können den Rückgabewert auswerten.
METHOD FB_Init: BOOL
VAR_INPUT    
bInitRetains: BOOL; // TRUE: Die Retain-Variablen werden initialisiert (Reset warm / Reset kalt)    
bInCopyCode: BOOL;  // TRUE: Die Instanz wird danach in den Kopiercode kopiert (Online-Change)
END_VAR
VAR
  tmp_udiResult     : SysTypes.RTS_IEC_RESULT;
  tmp_hEvent        : CmpEventMgr.RTS_IEC_HANDLE;
END_VAR
(* Open Event Com Cycle *)
HANDLE_EVENT_COM_CYCLE := CmpEventMgr_Implementation.EventOpen(CmpApp.EventIDs.EVT_CommCycle,cmpApp.EventIDs.CMPID_CmpApp,tmp_udiResult);
(* Self Register to the open event *)
HANDLE_CALBACK := CmpEventMgr.EventRegisterCallback(HANDLE_EVENT_COM_CYCLE, THIS^,tmp_udiResult);
(* Get Application *)
IF APPLICATION_THIS = 0 THEN
	APPLICATION_THIS 				:=	CmpApp.AppGetCurrent(ADR(RESULT_APPLICATION_THIS));
END_IF;
END_METHOD

//FB_Exit muss explizit implementiert werden. Wenn es eine Implementierung gibt, dann wird 
//die Methode aufgerufen, bevor die Steuerung den Code der Funktionsbaustein-Instanz entfernt
//(impliziter Aufruf. Der Rückgabewert wird nicht ausgewertet.
METHOD FB_Exit: BOOL
VAR_INPUT    
bInCopyCode: BOOL;  // TRUE: Die Exit-Methode wird aufgerufen, um die Instanz zu verlassen, die hinterher kopiert wird Online-Change).  
END_VAR
IF HANDLE_CYCLIC_TRENDLOG_BACKGROUND <> 0 THEN
	CmpIecTask.IecTaskDelete2(HANDLE_CYCLIC_TRENDLOG_BACKGROUND,0);
	HANDLE_CYCLIC_TRENDLOG_BACKGROUND := 0;
END_IF;
IF HANDLE_CYCLIC_TRENDLOG <> 0 THEN
	CmpIecTask.IecTaskDelete2(HANDLE_CYCLIC_TRENDLOG,0);
	HANDLE_CYCLIC_TRENDLOG := 0;
END_IF;
HANDLE_CYCLIC_TRENDLOG_BACKGROUND := 0;
HANDLE_CYCLIC_TRENDLOG := 0;

CmpEventMgr_Implementation.EventUnregisterCallback(hEvent := HANDLE_EVENT_COM_CYCLE, hInterface := HANDLE_CALBACK);
END_METHOD

{attribute 'm4export_hide'}
(* The interface ICmpEventCallback must be registered for an event. If this event is posted, this callback method is called.*)
METHOD EventCallback : SysTypes.RTS_IEC_RESULT
VAR_INPUT
	(*Pointer to the event parameters, see Struct EventParam*)
	pEventParam	: POINTER TO EventParam;
END_VAR
VAR
	IEC_RESULT		:	SysTypes.RTS_IEC_RESULT;
END_VAR
IF pEventParam^.CmpIdProvider = CmpApp.EventIDs.CMPID_CmpApp THEN
	IF pEventParam^.EventId = CmpApp.EventIDs.EVT_CommCycle THEN		
		(*----------------------SET CYCLIC BACKGROUND TASK PARAMETER--------------------------*)
		IF HANDLE_CYCLIC_TRENDLOG_BACKGROUND = 0 THEN
			NAME_CYCLIC_TRENDLOG_BACKGROUND									:= 'CYCLIC_TRENDLOG_BACKGROUND_CTA';
			INFO_CYCLIC_TRENDLOG_BACKGROUND.dwVersion						:= 2;
			INFO_CYCLIC_TRENDLOG_BACKGROUND.pszName 						:= ADR(NAME_CYCLIC_TRENDLOG_BACKGROUND);
			INFO_CYCLIC_TRENDLOG_BACKGROUND.bWatchdog						:= FALSE;
			INFO_CYCLIC_TRENDLOG_BACKGROUND.dwWatchdogSensitivity			:= 5;
			INFO_CYCLIC_TRENDLOG_BACKGROUND.dwWatchdogTime					:= 120000000;
			INFO_CYCLIC_TRENDLOG_BACKGROUND.nPriority						:= 15;
			INFO_CYCLIC_TRENDLOG_BACKGROUND.dwInterval						:= 500000;
			INFO_CYCLIC_TRENDLOG_BACKGROUND.dwEventFunctionPointer 			:= ADR(CYCLIC_TYPE);
			INFO_CYCLIC_TRENDLOG_BACKGROUND.dwTaskEntryFunctionPointer 		:= ADR(CYCLIC_TRENDLOG_BACKGROUND_CTA);
			INFO_CYCLIC_TRENDLOG_BACKGROUND.pszExternalEvent				:= ADR(EMPTY_STRING);
															
			HANDLE_CYCLIC_TRENDLOG_BACKGROUND := 	CmpIecTask.IecTaskCreate(	pApp				:= APPLICATION_THIS,
																				pTaskInfo			:= ADR(INFO_CYCLIC_TRENDLOG_BACKGROUND),											
																				pResult				:= ADR(RESULT_CYCLIC_TRENDLOG_BACKGROUND));
			IF RESULT_CYCLIC_TRENDLOG_BACKGROUND <> CmpErrors.Errors.ERR_OK THEN
				HANDLE_CYCLIC_TRENDLOG_BACKGROUND := 0;
			END_IF;														
		END_IF;		
		(*----------------------SET CYCLIC TRENDLOG TASK PARAMETER--------------------------*)
		IF HANDLE_CYCLIC_TRENDLOG = 0 THEN
			NAME_CYCLIC_TRENDLOG									:= 'CYCLIC_TRENDLOG_CTA';
			INFO_CYCLIC_TRENDLOG.dwVersion							:= 2;
			INFO_CYCLIC_TRENDLOG.pszName 							:= ADR(NAME_CYCLIC_TRENDLOG);
			INFO_CYCLIC_TRENDLOG.bWatchdog							:= FALSE;
			INFO_CYCLIC_TRENDLOG.dwWatchdogSensitivity				:= 5;
			INFO_CYCLIC_TRENDLOG.dwWatchdogTime						:= 120000000;
			INFO_CYCLIC_TRENDLOG.nPriority							:= 14;
			INFO_CYCLIC_TRENDLOG.dwInterval							:= 150000;
			INFO_CYCLIC_TRENDLOG.dwEventFunctionPointer 			:= ADR(CYCLIC_TYPE);
			INFO_CYCLIC_TRENDLOG.dwTaskEntryFunctionPointer 		:= ADR(CYCLIC_TRENDLOG_CTA);
			INFO_CYCLIC_TRENDLOG.pszExternalEvent					:= ADR(EMPTY_STRING);
															
			HANDLE_CYCLIC_TRENDLOG := 		CmpIecTask.IecTaskCreate(	pApp				:= APPLICATION_THIS,
																		pTaskInfo			:= ADR(INFO_CYCLIC_TRENDLOG),											
																		pResult				:= ADR(RESULT_CYCLIC_TRENDLOG));
			IF RESULT_CYCLIC_TRENDLOG <> CmpErrors.Errors.ERR_OK THEN
				HANDLE_CYCLIC_TRENDLOG := 0;
			END_IF;				
		END_IF;		
						
(*-----------------------------TASK Run Check---------------------------------------------*)
		IF APPLICATION_THIS <> 0 THEN
			IF APPLICATION_THIS^.udiState = CmpApp.AS_RUN THEN
				(* HANDLE_CYCLIC_BACKGROUND *)
				IF HANDLE_CYCLIC_TRENDLOG_BACKGROUND <> 0 THEN
					TEMP_TASK_INFO := CmpIecTask.IecTaskGetInfo3(HANDLE_CYCLIC_TRENDLOG_BACKGROUND,ADR(IEC_RESULT));
					IF TEMP_TASK_INFO <> 0 THEN
						IF TEMP_TASK_INFO^.pszName <> 0 AND INFO_CYCLIC_TRENDLOG_BACKGROUND.pszName <> 0 THEN 
							IF TEMP_TASK_INFO^.pszName^ = INFO_CYCLIC_TRENDLOG_BACKGROUND.pszName^ THEN
								(* Check if Valid *)
								IF INFO_CYCLIC_TRENDLOG_BACKGROUND.iState.0 = 0 THEN
									HANDLE_CYCLIC_TRENDLOG_BACKGROUND := CmpIecTask.IecTaskReload(HANDLE_CYCLIC_TRENDLOG_BACKGROUND,TO_UDINT(CmpiecTask.Timeout.RTS_TIMEOUT_DEFAULT),ADR(RESULT_CYCLIC_TRENDLOG_BACKGROUND));
								END_IF;
								(* Check if Suspended *)
								IF INFO_CYCLIC_TRENDLOG_BACKGROUND.iState.2 = 1 THEN
									HANDLE_CYCLIC_TRENDLOG_BACKGROUND := CmpIecTask.IecTaskReload(HANDLE_CYCLIC_TRENDLOG_BACKGROUND,TO_UDINT(CmpiecTask.Timeout.RTS_TIMEOUT_DEFAULT),ADR(RESULT_CYCLIC_TRENDLOG_BACKGROUND));
								END_IF;
								(* Check if Deletet *)
								IF INFO_CYCLIC_TRENDLOG_BACKGROUND.iState.3 = 1 THEN
									HANDLE_CYCLIC_TRENDLOG_BACKGROUND := CmpIecTask.IecTaskReload(HANDLE_CYCLIC_TRENDLOG_BACKGROUND,TO_UDINT(CmpiecTask.Timeout.RTS_TIMEOUT_DEFAULT),ADR(RESULT_CYCLIC_TRENDLOG_BACKGROUND));
								END_IF;
							ELSE
								HANDLE_CYCLIC_TRENDLOG_BACKGROUND := 0;
							END_IF;	
						ELSE
							HANDLE_CYCLIC_TRENDLOG_BACKGROUND := 0;
						END_IF;
					ELSE
						HANDLE_CYCLIC_TRENDLOG_BACKGROUND := 0;	
					END_IF;
				END_IF;
				(* HANDLE_CYCLIC_TRENDLOG *)
				IF HANDLE_CYCLIC_TRENDLOG <> 0 THEN
					TEMP_TASK_INFO := CmpIecTask.IecTaskGetInfo3(HANDLE_CYCLIC_TRENDLOG,ADR(IEC_RESULT));
					IF TEMP_TASK_INFO <> 0 THEN
						IF TEMP_TASK_INFO^.pszName <> 0 AND INFO_CYCLIC_TRENDLOG.pszName <> 0 THEN 
							IF TEMP_TASK_INFO^.pszName^ = INFO_CYCLIC_TRENDLOG.pszName^ THEN					
								(* Check IF Valid *)
								IF INFO_CYCLIC_TRENDLOG.iState.0 = 0 THEN
									HANDLE_CYCLIC_TRENDLOG := CmpIecTask.IecTaskReload(HANDLE_CYCLIC_TRENDLOG,TO_UDINT(CmpiecTask.Timeout.RTS_TIMEOUT_DEFAULT),ADR(RESULT_CYCLIC_TRENDLOG));
								END_IF;
								(* Check if Suspended *)
								IF INFO_CYCLIC_TRENDLOG.iState.2 = 1 THEN
									HANDLE_CYCLIC_TRENDLOG := CmpIecTask.IecTaskReload(HANDLE_CYCLIC_TRENDLOG,TO_UDINT(CmpiecTask.Timeout.RTS_TIMEOUT_DEFAULT),ADR(RESULT_CYCLIC_TRENDLOG));
								END_IF;
								(* Check if Deletet *)
								IF INFO_CYCLIC_TRENDLOG.iState.3 = 1 THEN
									HANDLE_CYCLIC_TRENDLOG := CmpIecTask.IecTaskReload(HANDLE_CYCLIC_TRENDLOG,TO_UDINT(CmpiecTask.Timeout.RTS_TIMEOUT_DEFAULT),ADR(RESULT_CYCLIC_TRENDLOG));
								END_IF;
							ELSE
								HANDLE_CYCLIC_TRENDLOG := 0;
							END_IF;	
						ELSE
							HANDLE_CYCLIC_TRENDLOG := 0;
						END_IF;
					ELSE
						HANDLE_CYCLIC_TRENDLOG := 0;	
					END_IF;								
				END_IF;
			END_IF;		
		END_IF;		
	END_IF;
END_IF;
END_METHOD

END_FUNCTION_BLOCK

// 30 Program Organization Units/TASK_SCHEDULER/CYCLIC_TRENDLOG_BACKGROUND_CTA
FUNCTION CYCLIC_TRENDLOG_BACKGROUND_CTA : BOOL
VAR_INPUT
    parameter : IEC_CYCLE_STRUCT;
END_VAR
VAR
    udiState : UDINT;
    hTask	 : SysTypes.RTS_IEC_HANDLE;
	dwOldSema	: DWORD;
END_VAR

(* ----- mandatory cyclic task frame code begin ----- *)
udiState := parameter.pApplication^.udiState;
hTask := parameter.hTaskHandle;
IF udiState = CmpApp.AS_STOP THEN
    RETURN;
END_IF;
IF parameter.pTaskInfo^.bWatchdog THEN
    IecTaskEnableWatchdog(hTask);
END_IF;
IF udiState = CmpApp.AS_RUN OR udiState = CmpApp.AS_SINGLE_CYCLE OR udiState = CmpApp.AS_DEBUG_STEP THEN
	dwOldSema := TEST_AND_SET(GVL_TREND_TASK_PROVIDER.dwSEMA_BACK);
	IF dwOldSema = 0 THEN
		GVL_TREND.ASYNC_SEND();
		parameter.pTaskInfo^.dwIECCycleCount := parameter.pTaskInfo^.dwIECCycleCount + 1;
		GVL_TREND_TASK_PROVIDER.dwSEMA_BACK := 0;
	END_IF;
END_IF
(* ------ mandatory cyclic task frame code end ------ *)

END_FUNCTION

// 30 Program Organization Units/TASK_SCHEDULER/CYCLIC_TRENDLOG_CTA
FUNCTION CYCLIC_TRENDLOG_CTA : BOOL
VAR_INPUT
    parameter : IEC_CYCLE_STRUCT;
END_VAR
VAR
    udiState 	: UDINT;
    hTask 		: SysTypes.RTS_IEC_HANDLE;
	dwOldSema	: DWORD;
END_VAR

(* ----- mandatory cyclic task frame code begin ----- *)
udiState := parameter.pApplication^.udiState;
hTask := parameter.hTaskHandle;
IF udiState = CmpApp.AS_STOP THEN
    RETURN;
END_IF;
IF parameter.pTaskInfo^.bWatchdog THEN
    IecTaskEnableWatchdog(hTask);
END_IF;
IF udiState = CmpApp.AS_RUN OR udiState = CmpApp.AS_SINGLE_CYCLE OR udiState = CmpApp.AS_DEBUG_STEP  THEN
	dwOldSema := TEST_AND_SET(GVL_TREND_TASK_PROVIDER.dwSEMA_CYCLIC);
	IF dwOldSema = 0 THEN
		GVL_TREND.FB_INFLUX_LOG_OBJ();
		parameter.pTaskInfo^.dwIECCycleCount := parameter.pTaskInfo^.dwIECCycleCount + 1;
		GVL_TREND_TASK_PROVIDER.dwSEMA_CYCLIC := 0;
	END_IF;
END_IF
(* ------ mandatory cyclic task frame code end ------ *)

END_FUNCTION

// 40 Visualizations/visInfluxDb
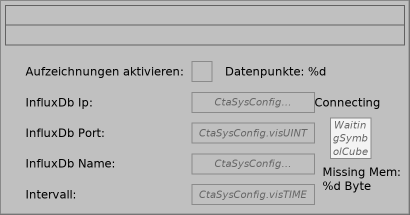
VISUALIZATION visInfluxDb  // 410x215
    Frame (0,0 410x215)
        shows visInfluxDbTemp(FB_INFLUX_LOG := GVL_TREND.FB_INFLUX_LOG_OBJ, FB_NODE_FACTORY := GVL_TREND.FB_INFLUX_NODE_FACTORY)
END_VISUALIZATION

// 40 Visualizations/visInfluxDbTemp
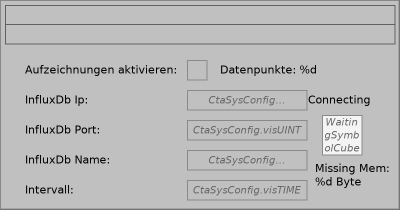
VISUALIZATION visInfluxDbTemp  // 400x210
VAR_IN_OUT
	FB_INFLUX_LOG	:	FB_INFLUX_LOG;
	FB_NODE_FACTORY	:	FB_NODE_FACTORY;
END_VAR
    RoundedRectangle (0,0 400x210)
    Textfield (5,5 390x20), text list: 'InfluxStartup', text index: FB_INFLUX_LOG.usiStartUpCase
    Textfield (5,24 390x20), text list: 'LogState', text index: FB_INFLUX_LOG.usiLogCase
    Label (22,120 100x20), "InfluxDb Port:"
    Label (22,90 100x20), "InfluxDb Ip:"
    Label (22,150 100x20), "InfluxDb Name:"
    Group (312,90 80x65), invisible if: FB_INFLUX_LOG.usiStartUpCase = 2
        WaitingSymbolCube (10,25 40x40), invisible if: FB_INFLUX_LOG.usiStartUpCase = 2
        Label (0,0 55x20), "Connecting", invisible if: FB_INFLUX_LOG.usiStartUpCase = 2
    Label (22,180 120x20), "Intervall:"
    Frame (187,180 120x20)
        shows CtaSysConfig.visTIME(visfbTIMEIn := FB_INFLUX_LOG.scParameter.fbtLogIntervall)
    Frame (187,150 120x20)
        shows CtaSysConfig.visSTRING40(visfbSTRING40In := FB_INFLUX_LOG.scParameter.fbDataBase)
    Frame (187,90 120x20)
        shows CtaSysConfig.visSTRING40(visfbSTRING40In := FB_INFLUX_LOG.scParameter.fbServerIp)
    Frame (187,120 120x20)
        shows CtaSysConfig.visUINT(visfbUINTIn := FB_INFLUX_LOG.scParameter.fbuiPort)
    Frame (187,60 20x20)
        shows CtaSysConfig.visBOOL(visfbBOOLIn := FB_INFLUX_LOG.scParameter.fbxEnable)
    Label (22,60 160x20), "Aufzeichnungen aktivieren:"
    Textfield (217,60 178x20), "Datenpunkte: %d", text variable: FB_INFLUX_LOG._COUNT
    Textfield (312,150 83x50), "Missing Mem: %d Byte", text variable: TO_ULINT(FB_NODE_FACTORY.udiMissingBoolMemory + FB_NODE_FACTORY.udiMissingIntMemory + FB_NODE_FACTORY.udiMissingRealMemory + FB_NODE_FACTORY.udiMissingStringMemory), invisible if: TO_ULINT(FB_NODE_FACTORY.udiMissingBoolMemory + FB_NODE_FACTORY.udiMissingIntMemory + FB_NODE_FACTORY.udiMissingRealMemory + FB_NODE_FACTORY.udiMissingStringMemory) = 0
END_VISUALIZATION

// 40 Visualizations/VIS_POPUP_INFLUXDB
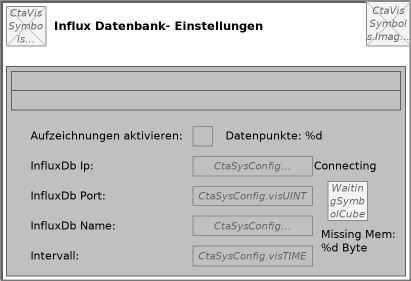
VISUALIZATION VIS_POPUP_INFLUXDB  // 411x281
    RoundedRectangle (1,1 410x280)
    Image (6,6 40x40), image: CtaVisSymbols.ImagePool.InfluxDb_Logo
    Image (366,1 45x45), image: CtaVisSymbols.ImagePool.close_solo_black
        OnMouseClick:  Dialog=Current Dialog, Result=None, NumpadKeypadSet=True
    Frame (6,66 400x210)
        shows visInfluxDb()
    Label (51,16 300x20), "Influx Datenbank- Einstellungen"
    InvisibleInput (1,1 365x45)
END_VISUALIZATION

(* text list InfluxStartup (id | default)
  0 | Database state: initializing
  1 | Database state: creating database
  2 | Database state: database created
   |  *)

(* text list LogState (id | default)
  0 | Log Status: waiting for database
  1 | Log Status: opening file
  2 | Log Status: logging
  3 | Log Status: closing and sending file
   |  *)
